(* IEC 61131-3 sources: POMIRTS_lab3/AS/Library/LoopConR/V2.80.0, 3 files *)

(* ---- LoopConR.typ ---- *)
TYPE
	lcrCurveByPoints_TabEntry_type : 	STRUCT
		x : REAL;
		y : REAL;
	END_STRUCT;
	lcrdblpid_par_typ : 	STRUCT
		Y_max : REAL;
		Y_min : REAL;
		K_fact : INT;
		Kp : REAL;
		Tn : REAL;
		Tv : REAL;
	END_STRUCT;
	lcrdblpid_tune_typ : 	STRUCT
		P1_manualAdjust : INT;
		I1_manualAdjust : INT;
		D1_manualAdjust : INT;
		P2_manualAdjust : INT;
		I2_manualAdjust : INT;
		D2_manualAdjust : INT;
		X_min : REAL;
		X_max : REAL;
		X0 : REAL;
		de_min : REAL;
		Y0 : REAL;
		Y1step : REAL;
		Y2step : REAL;
		tuneY1_opt : UDINT;
		tuneY2_opt : UDINT;
		tune_first : USINT;
		hyst : REAL;
		measDelta : REAL;
		osc_opt : lcrpid_tune_osc_options_typ;
		step_opt : lcrpid_tune_step_options_typ;
	END_STRUCT;
	lcrpid_internal_typ : 	STRUCT
		size : UINT;
		valid : BOOL;
		WX_max : REAL;
		WX_min : REAL;
		invert : BOOL;
		deadband : REAL;
		deadband_mode : USINT;
		dY_max : REAL;
		Kp : REAL;
		Kp_Tn : REAL;
		Tv_Tf : REAL;
		Tf_reciproc : REAL;
		Kw : REAL;
		Kfbk_Kp : REAL;
		Kfbk_Kp_max : REAL;
		fbk_mode : USINT;
		d_mode : USINT;
		force_mode : USINT;
		Y_force : REAL;
		W : REAL;
		X : REAL;
		pid_init : USINT;
		Yp1 : DINT;
		Yp2 : DINT;
		dYi1 : DINT;
		dYi2 : DINT;
		Yi1 : DINT;
		Yi2 : DINT;
		dt_Tf : REAL;
		a11 : DINT;
		a12 : DINT;
		a21 : DINT;
		a22 : DINT;
		Yd1 : DINT;
		Yd2 : DINT;
		Ytotal1 : DINT;
		Ytotal2 : DINT;
		Ylim1 : DINT;
		Ylim2 : DINT;
		Y1 : DINT;
		Y2 : DINT;
		deltaY_fbk : REAL;
		e_fbk : REAL;
	END_STRUCT;
	lcrpid_old_typ : 	STRUCT
		processPar : lcrpid_procPar_typ;
		P_manualAdjust : INT;
		I_manualAdjust : INT;
		D_manualAdjust : INT;
		Y_min : REAL;
		Y_max : REAL;
		dY_max : REAL;
		Tf_Tv : REAL;
		Kw : REAL;
		Kfbk : REAL;
		deadband : REAL;
		W : REAL;
		request : UDINT;
		fbk_mode : USINT;
		d_mode : USINT;
		invert : BOOL;
		enable : BOOL;
	END_STRUCT;
	lcrpid_osc_per_typ : 	STRUCT
		max : lcrpid_osc_val_typ;
		min : lcrpid_osc_val_typ;
	END_STRUCT;
	lcrpid_osc_val_typ : 	STRUCT
		X : REAL;
		t : REAL;
	END_STRUCT;
	lcrpid_procPar_typ : 	STRUCT
		size : UINT;
		valid : BOOL;
		stepResp_valid : BOOL;
		stepResp_v : REAL;
		stepResp_t_u : REAL;
		stepResp_t_g : REAL;
		osc_valid : BOOL;
		osc_amplitudeRatio : REAL;
		osc_tPeriod : REAL;
		force_params : BOOL;
		Kp : REAL;
		Kp_tune : REAL;
		Tn : REAL;
		Tn_tune : REAL;
		Tv : REAL;
		Tv_tune : REAL;
	END_STRUCT;
	lcrpid_tune_addpar_typ : 	STRUCT
		t_max_tune : REAL;
		WX_min : REAL;
		WX_max : REAL;
		dY_max : REAL;
		Tf_Tv : REAL;
		Kw : REAL;
		Kfbk : REAL;
		fbk_mode : USINT;
		d_mode : USINT;
		deadband : REAL;
		deadband_mode : USINT;
		invert : BOOL;
	END_STRUCT;
	lcrpid_tune_osc_options_typ : 	STRUCT
		osc_minAmplitude : REAL;
		Q_min : REAL;
	END_STRUCT;
	lcrpid_tune_osc_typ : 	STRUCT
		options : lcrpid_tune_osc_options_typ;
		oscPhase : UINT;
		dir : SINT;
		enHi : BOOL;
		enLo : BOOL;
		Y_hi : REAL;
		Y_lo : REAL;
		i_maxPeriod : UINT;
		i_period : UINT;
		X_ampl : REAL;
		X_avg : REAL;
		X_min_avg : REAL;
		X_max_avg : REAL;
		Y_avg : REAL;
		deltaY : REAL;
		t_Ylohi : ARRAY[0..4] OF REAL;
		t_Yhilo : ARRAY[0..4] OF REAL;
		Q_act : REAL;
		a_wx : REAL;
		amplitudeRatio : REAL;
		Ku : REAL;
		tPeriod : REAL;
		period : ARRAY[0..4] OF lcrpid_osc_per_typ;
	END_STRUCT;
	lcrpid_tune_step_options_typ : 	STRUCT
		eqDeltaX : REAL;
		eqDeltaWX : REAL;
		eqDeltat : REAL;
		evalDeltaX : REAL;
		evalNfilter : UINT;
		exitNotMaxdXCount : UINT;
		exitdXRatio : REAL;
	END_STRUCT;
	lcrpid_tune_step_typ : 	STRUCT
		options : lcrpid_tune_step_options_typ;
		Y0 : REAL;
		Y1 : REAL;
		t_jump : REAL;
		W : REAL;
		X0 : REAL;
		Xmax : REAL;
		Xmin : REAL;
		Xfiltered : REAL;
		deltaXok : BOOL;
		deltaWXok : BOOL;
		eqTime : REAL;
		dir : SINT;
		deltaX : REAL;
		X1 : REAL;
		t1 : REAL;
		t1set : BOOL;
		dX_dt : REAL;
		dX_dt_max : REAL;
		XmaxGrad : REAL;
		maxX1 : REAL;
		maxX2 : REAL;
		maxt1 : REAL;
		maxt2 : REAL;
		tmaxGrad : REAL;
		gainFactor : REAL;
		deadTime : REAL;
		riseTime : REAL;
		notMaxCount : UINT;
		gradientRatio : REAL;
	END_STRUCT;
	lcrpt2o_Internal_typ : 	STRUCT
		Ts : DINT;
		Ts_dbl_1 : UDINT;
		Ts_dbl_2 : UDINT;
		V_old : REAL;
		D_old : REAL;
		Tf_old : REAL;
		Set_y_old : USINT;
		Set_y_2 : USINT;
		x1_dbl_1 : UDINT;
		x1_dbl_2 : UDINT;
		x2_dbl_1 : UDINT;
		x2_dbl_2 : UDINT;
		Sqrt_D_1_dbl_1 : UDINT;
		Sqrt_D_1_dbl_2 : UDINT;
		Ts_Tf_dbl_1 : UDINT;
		Ts_Tf_dbl_2 : UDINT;
		Exp_D_Ts_Tf_dbl_1 : UDINT;
		Exp_D_Ts_Tf_dbl_2 : UDINT;
		a0_dbl_1 : UDINT;
		a0_dbl_2 : UDINT;
		a1_dbl_1 : UDINT;
		a1_dbl_2 : UDINT;
		b0_dbl_1 : UDINT;
		b0_dbl_2 : UDINT;
		b1_dbl_1 : UDINT;
		b1_dbl_2 : UDINT;
		Bootkey : UDINT;
	END_STRUCT;
	lcrschedule_add_typ : 	STRUCT
		periodTime : REAL;
		onTime : REAL;
		t_on_intern : REAL;
		bcOnTime : REAL;
		sortIndex : UINT;
		fbkPWM : LCRPWM;
		flagDelay : BOOL;
	END_STRUCT;
	lcrschedule_par_typ : 	STRUCT
		P : REAL;
		X : REAL;
		pulse : BOOL;
		Pout : REAL;
		lim : BOOL;
		Internal : lcrschedule_add_typ;
	END_STRUCT;
	lcrslimpid_par_typ : 	STRUCT
		Y_max : REAL;
		Y_min : REAL;
		Kp : REAL;
		Tn : REAL;
		Tv : REAL;
		Kfbk : REAL;
	END_STRUCT;
	lcrtemp_add_typ : 	STRUCT
		mem01 : REAL;
		mem02 : REAL;
		mem10 : REAL;
		mem20 : REAL;
		exp_mem : REAL;
		cnt01 : REAL;
		cnt02 : REAL;
		cnt10 : REAL;
		cnt20 : REAL;
		cnt03 : REAL;
		cnt30 : REAL;
		cnt00 : REAL;
		t_ignore_dT_heat : REAL;
		t_ignore_dT_free : REAL;
		t_ignore_dT_cool : REAL;
		yMin : REAL;
		yMax : REAL;
		reserved3 : UDINT;
		reserved4 : UDINT;
		reserved5 : BOOL;
		reserved6 : BOOL;
	END_STRUCT;
	lcrtemp_pid_internal_typ : 	STRUCT
		enable_cooling : BOOL;
		disable_heating : BOOL;
		hyst : REAL;
		delay : REAL;
		Kw : REAL;
		Kfbk : REAL;
		Kp_h : REAL;
		Tn_h : REAL;
		Tv_h : REAL;
		Kp_c : REAL;
		Tn_c : REAL;
		Tv_c : REAL;
		dynGeneral : REAL;
		dynHeat : REAL;
		dynCool : REAL;
		mem01 : REAL;
		mem02 : REAL;
		mem10 : REAL;
		mem20 : REAL;
		exp_mem : REAL;
		yMin : REAL;
		yMax : REAL;
	END_STRUCT;
	lcrtemp_pid_opt_typ : 	STRUCT
		Kp_h : REAL;
		Tn_h : REAL;
		Tv_h : REAL;
		Kp_c : REAL;
		Tn_c : REAL;
		Tv_c : REAL;
		dynGeneral : REAL;
		dynHeat : REAL;
		dynCool : REAL;
	END_STRUCT;
	lcrtemp_pid_set_typ : 	STRUCT
		hyst : REAL;
		delay : REAL;
		Kw : REAL;
		Kfbk : REAL;
	END_STRUCT;
	lcrtemp_set_typ : 	STRUCT
		enable_cooling : BOOL;
		disable_heating : BOOL;
		PIDpara : lcrtemp_pid_opt_typ;
		TuneSet : lcrtemp_tune_set_typ;
		PIDSet : lcrtemp_pid_set_typ;
		Internal : lcrtemp_add_typ;
	END_STRUCT;
	lcrtemp_tune_internal_typ : 	STRUCT
		cool_tuning : BOOL;
		disable_heating : BOOL;
		mode : UDINT;
		Temp_amb : REAL;
		dRatio_heat : REAL;
		cnt_tp_heat : REAL;
		delta_T_heat : REAL;
		dT_min_heat : REAL;
		dRatio_free : REAL;
		cnt_tp_free : REAL;
		delta_T_free : REAL;
		dT_min_free : REAL;
		dRatio_cool : REAL;
		cnt_tp_cool : REAL;
		delta_T_cool : REAL;
		dT_min_cool : REAL;
		delta_T_sync_heat : REAL;
		delta_dT_sync_heat : REAL;
		cnt_wait_heat : REAL;
		delta_T_sync_free : REAL;
		delta_dT_sync_free : REAL;
		cnt_wait_free : REAL;
		delta_T_sync_cool : REAL;
		delta_dT_sync_cool : REAL;
		cnt_wait_cool : REAL;
		filter_base_T : REAL;
		t_ignore_dT_heat : REAL;
		t_ignore_dT_free : REAL;
		t_ignore_dT_cool : REAL;
		delta_T_sync_stop : REAL;
	END_STRUCT;
	lcrtemp_tune_set_typ : 	STRUCT
		mode : UDINT;
		Temp_amb : REAL;
		dRatio_heat : REAL;
		cnt_tp_heat : REAL;
		delta_T_heat : REAL;
		dT_min_heat : REAL;
		dRatio_free : REAL;
		cnt_tp_free : REAL;
		delta_T_free : REAL;
		dT_min_free : REAL;
		dRatio_cool : REAL;
		cnt_tp_cool : REAL;
		delta_T_cool : REAL;
		dT_min_cool : REAL;
		delta_T_sync_heat : REAL;
		delta_dT_sync_heat : REAL;
		cnt_wait_heat : REAL;
		delta_T_sync_free : REAL;
		delta_dT_sync_free : REAL;
		cnt_wait_free : REAL;
		delta_T_sync_cool : REAL;
		delta_dT_sync_cool : REAL;
		cnt_wait_cool : REAL;
		filter_base_T : REAL;
		delta_T_sync_stop : REAL;
		Y_heat_tune : REAL;
	END_STRUCT;
END_TYPE

(* ---- LoopConR.fun ---- *)
FUNCTION_BLOCK LCRPID
	VAR_INPUT
		enable : BOOL;
		ident : UDINT;
		W : REAL;
		X : REAL;
		Y_max : REAL;
		Y_min : REAL;
		A : REAL;
		Y_man : REAL;
		Y_fbk : REAL;
		hold_I : BOOL;
		mode : USINT;
	END_VAR
	VAR_OUTPUT
		status : UINT;
		e : REAL;
		Y : REAL;
		Yp : REAL;
		Yi : REAL;
		Yd : REAL;
	END_VAR
	VAR
		Set_Yi : BOOL;
		Yi_set : REAL;
		force_Yi : BOOL;
		Yi_min : REAL;
		Yi_max : REAL;
		joltFreeDoneLowerLim : BOOL;
		joltFreeDoneUpperLim : BOOL;
		Yi_minInternal : REAL;
		Yi_maxInternal : REAL;
		Tv_Tf_old : REAL;
		enable_old : BOOL;
		e_old : REAL;
		deadband_state : UINT;
		sysinfo_inst : SysInfo;
		scal_inst : LCRScal;
		store1 : UDINT;
		store2 : UDINT;
		timeCnt : UDINT;
		musecs_old : UINT;
	END_VAR
END_FUNCTION_BLOCK

FUNCTION_BLOCK LCRScal
	VAR_INPUT
		x : REAL;
		x1 : REAL;
		y1 : REAL;
		x2 : REAL;
		y2 : REAL;
	END_VAR
	VAR_OUTPUT
		y : REAL;
	END_VAR
END_FUNCTION_BLOCK

FUNCTION_BLOCK LCRCurveByPoints
	VAR_INPUT
		x : REAL;
		NoOfPoints : UINT;
		ptr_table : REFERENCE TO lcrCurveByPoints_TabEntry_type;
	END_VAR
	VAR_OUTPUT
		status : UINT;
		y : REAL;
	END_VAR
	VAR
		i_tab : INT;
		iterations : UINT;
		scal1 : LCRScal;
	END_VAR
END_FUNCTION_BLOCK

FUNCTION_BLOCK LCRPIDpara
	VAR_INPUT
		enable : BOOL;
		enter : BOOL;
		WX_max : REAL;
		WX_min : REAL;
		invert : BOOL;
		deadband : REAL;
		deadband_mode : USINT;
		dY_max : REAL;
		Kp : REAL;
		Tn : REAL;
		Tv : REAL;
		Tf : REAL;
		Kw : REAL;
		Kfbk : REAL;
		fbk_mode : USINT;
		d_mode : USINT;
	END_VAR
	VAR_OUTPUT
		status : UINT;
		ident : UDINT;
	END_VAR
	VAR
		internal_data : lcrpid_internal_typ;
	END_VAR
END_FUNCTION_BLOCK

FUNCTION_BLOCK LCRContinServo
	VAR_INPUT
		enable : BOOL;
		x : REAL;
		max_value : REAL;
		min_value : REAL;
		t_impulse : REAL;
		t_change_up : REAL;
		t_change_down : REAL;
		ref : BOOL;
	END_VAR
	VAR_OUTPUT
		status : UINT;
		up : BOOL;
		down : BOOL;
		hysteresis_up : REAL;
		hysteresis_down : REAL;
		refOk : BOOL;
	END_VAR
	VAR
		enable_old : BOOL;
		counter_state : UINT;
		bootkey_old : UDINT;
		systicks_old : UDINT;
		musecs_old : UINT;
		ref_old : BOOL;
		t_cnt_1 : DINT;
		t_cnt_2 : DINT;
		y_dbl_1 : DINT;
		y_dbl_2 : DINT;
		sysInfo_inst : SysInfo;
	END_VAR
END_FUNCTION_BLOCK

FUNCTION_BLOCK LCRPT1
	VAR_INPUT
		enable : BOOL;
		x : REAL;
		t : REAL;
		y_set : REAL;
		set : BOOL;
	END_VAR
	VAR_OUTPUT
		status : UINT;
		y : REAL;
	END_VAR
	VAR
		counter_state : UINT;
		bootkey_old : UDINT;
		systicks_old : UDINT;
		musecs_old : UINT;
		y_dbl_1 : DINT;
		y_dbl_2 : DINT;
		sysinfo_inst : SysInfo;
	END_VAR
END_FUNCTION_BLOCK

FUNCTION_BLOCK LCRRamp
	VAR_INPUT
		enable : BOOL;
		x : REAL;
		dy_up : REAL;
		dy_down : REAL;
		y_max : REAL;
		y_min : REAL;
		y_set : REAL;
		set : BOOL;
	END_VAR
	VAR_OUTPUT
		status : UINT;
		y : REAL;
		x_reached : BOOL;
		max_limit : BOOL;
		min_limit : BOOL;
	END_VAR
	VAR
		y_dbl_1 : DINT;
		y_dbl_2 : DINT;
		timestore1 : UDINT;
		timestore2 : UDINT;
		getDtForceOff : UDINT;
		sysinfo_inst : SysInfo;
	END_VAR
END_FUNCTION_BLOCK

FUNCTION_BLOCK LCRIntegrate
	VAR_INPUT
		enable : BOOL;
		x : REAL;
		tn : REAL;
		y_max : REAL;
		y_min : REAL;
		y_set : REAL;
		set : BOOL;
	END_VAR
	VAR_OUTPUT
		status : UINT;
		y : REAL;
		max_limit : BOOL;
		min_limit : BOOL;
	END_VAR
	VAR
		counter_state : UINT;
		bootkey_old : UDINT;
		systicks_old : UDINT;
		musecs_old : UINT;
		y_dbl_1 : DINT;
		y_dbl_2 : DINT;
		sysinfo_inst : SysInfo;
	END_VAR
END_FUNCTION_BLOCK

FUNCTION_BLOCK LCRLimit
	VAR_INPUT
		in : REAL;
		max_value : DINT;
		min_value : DINT;
	END_VAR
	VAR_OUTPUT
		status : UINT;
		out : DINT;
		max_limit : BOOL;
		min_limit : BOOL;
	END_VAR
END_FUNCTION_BLOCK

FUNCTION_BLOCK LCRLimScal
	VAR_INPUT
		x : REAL;
		x1 : REAL;
		y1 : REAL;
		x2 : REAL;
		y2 : REAL;
	END_VAR
	VAR_OUTPUT
		y : REAL;
	END_VAR
END_FUNCTION_BLOCK

FUNCTION_BLOCK LCRPWM
	VAR_INPUT
		enable : BOOL;
		x : REAL;
		max_value : REAL;
		min_value : REAL;
		t_min_pulse : REAL;
		t_period : REAL;
	END_VAR
	VAR_OUTPUT
		status : UINT;
		pulse : BOOL;
		t_on : REAL;
		t_off : REAL;
	END_VAR
	VAR
		cnt_terron_1 : DINT;
		cnt_terron_2 : DINT;
		cnt_terroff_1 : DINT;
		cnt_terroff_2 : DINT;
		cnt_t_pulse_1 : DINT;
		cnt_t_pulse_2 : DINT;
		store1 : UDINT;
		store2 : UDINT;
		timeCnt : UDINT;
		sysinfo_inst : SysInfo;
		corr : BOOL;
	END_VAR
END_FUNCTION_BLOCK

FUNCTION_BLOCK LCRMovAvgFlt
	VAR_INPUT
		enable : BOOL;
		x : REAL;
		base : UINT;
	END_VAR
	VAR_OUTPUT
		status : UINT;
		y : REAL;
	END_VAR
	VAR
		sum_old_dbl_1 : DINT;
		sum_old_dbl_2 : DINT;
		x_old : ARRAY[0..31] OF REAL;
		p_xold : UDINT;
		i_xold : UINT;
		base_old : UINT;
		enable_old : BOOL;
		bootkey_old : UDINT;
	END_VAR
END_FUNCTION_BLOCK

FUNCTION_BLOCK LCRTimeBasedOnOff
	VAR_INPUT
		enable : BOOL;
		x : REAL;
		max_value : REAL;
		min_value : REAL;
		timpulse : REAL;
		tchange_up : REAL;
		tchange_down : REAL;
		ref : BOOL;
	END_VAR
	VAR_OUTPUT
		status : UINT;
		up : BOOL;
		down : BOOL;
		hysteresis_up : REAL;
		hysteresis_down : REAL;
		refOk : BOOL;
	END_VAR
	VAR
		enable_old : BOOL;
		counter_state : UINT;
		bootkey_old : UDINT;
		systicks_old : UDINT;
		musecs_old : UINT;
		ref_old : BOOL;
		t_cnt_1 : DINT;
		t_cnt_2 : DINT;
		y_dbl_1 : DINT;
		y_dbl_2 : DINT;
		sysInfo_inst : SysInfo;
	END_VAR
END_FUNCTION_BLOCK

FUNCTION_BLOCK LCRDifferentiate
	VAR_INPUT
		enable : BOOL;
		x : REAL;
		tv : REAL;
		tf : REAL;
	END_VAR
	VAR_OUTPUT
		status : UINT;
		y : REAL;
	END_VAR
	VAR
		store1 : UDINT;
		store2 : UDINT;
		timeCnt : UDINT;
		counter_state : UINT;
		bootkey_old : UDINT;
		systicks_old : UDINT;
		musecs_old : UINT;
		sysinfo_inst : SysInfo;
		a11 : DINT;
		a12 : DINT;
		a21 : DINT;
		a22 : DINT;
	END_VAR
END_FUNCTION_BLOCK

FUNCTION_BLOCK LCRSlimPID
	VAR_INPUT
		enable : BOOL;
		W : REAL;
		X : REAL;
		request : UDINT;
		pPar : REFERENCE TO lcrslimpid_par_typ;
	END_VAR
	VAR_OUTPUT
		e : REAL;
		Y : REAL;
		status : UINT;
		addInfo : UINT;
	END_VAR
	VAR
		MovAvgFlt_inst : LCRMovAvgFlt;
		PIDTune_inst : LCRPIDTune;
		PID_inst : LCRPID;
		enable_old : BOOL;
		requ_old : UDINT;
	END_VAR
END_FUNCTION_BLOCK

FUNCTION_BLOCK LCRPIDTune
	VAR_INPUT
		enable : BOOL;
		Y_min : REAL;
		Y_max : REAL;
		Y0 : REAL;
		Y1 : REAL;
		okToStep : BOOL;
		X0 : REAL;
		X_min : REAL;
		X_max : REAL;
		P_manualAdjust : INT;
		I_manualAdjust : INT;
		D_manualAdjust : INT;
		request : UDINT;
		pAddPar : REFERENCE TO lcrpid_tune_addpar_typ;
		pOptions_osc : REFERENCE TO lcrpid_tune_osc_options_typ;
		pOptions_step : REFERENCE TO lcrpid_tune_step_options_typ;
	END_VAR
	VAR_OUTPUT
		status : UINT;
		addInfo : UINT;
		ident : UDINT;
		state : UINT;
		rdyToStep : BOOL;
	END_VAR
	VAR
		t_autotune : REAL;
		status_tmp : UINT;
		counter_state : UINT;
		bootkey_old : UDINT;
		systicks_old : UDINT;
		musecs_old : UINT;
		curveDown : BOOL;
		e : REAL;
		e_minAmp : REAL;
		e_old_up : REAL;
		e_old_down : REAL;
		curveUp : BOOL;
		e_old : REAL;
		sysinfo_inst : SysInfo;
		MovAvgFlt_inst : LCRMovAvgFlt;
		old : lcrpid_old_typ;
		processPar : lcrpid_procPar_typ;
		internal_data : lcrpid_internal_typ;
		addPar : lcrpid_tune_addpar_typ;
		oscillation : lcrpid_tune_osc_typ;
		stepresponse : lcrpid_tune_step_typ;
	END_VAR
END_FUNCTION_BLOCK

FUNCTION_BLOCK LCRPFM
	VAR_INPUT
		enable : BOOL;
		x : REAL;
		max_value : REAL;
		min_value : REAL;
		t_pulse : REAL;
		t_pause : REAL;
	END_VAR
	VAR_OUTPUT
		status : UINT;
		pulse : BOOL;
	END_VAR
	VAR
		area : REAL;
		area_c : REAL;
		range : REAL;
		last : REAL;
		tpls : REAL;
		enable_old : BOOL;
		counter_state : UINT;
		bootkey_old : UDINT;
		systicks_old : UDINT;
		musecs_old : UINT;
		sysinfo_inst : SysInfo;
	END_VAR
END_FUNCTION_BLOCK

FUNCTION_BLOCK LCRSimModExt
	VAR_INPUT
		enable : BOOL;
		Tt_h : DINT;
		Tt_c : DINT;
		k_h : REAL;
		k_c : REAL;
		PT2_T1 : REAL;
		PT2_T2 : REAL;
		Temp_amb : REAL;
		Temp_c : REAL;
		Alpha_h : REAL;
		Alpha_c : REAL;
	END_VAR
	VAR_OUTPUT
		y : REAL;
		status : UINT;
	END_VAR
	VAR
		Tt_heat : LCRTt;
		Tt_cool : LCRTt;
		k_h_intern : REAL;
		k_c_intern : REAL;
		PT2 : LCRPT2;
		y_c : REAL;
		y_end : REAL;
		y_h : REAL;
		Bootkey : UDINT;
		enable_old : BOOL;
	END_VAR
END_FUNCTION_BLOCK

FUNCTION_BLOCK LCRTt
	VAR_INPUT
		enable : BOOL;
		Tt : DINT;
		x : REAL;
		y_set : REAL;
		set : BOOL;
	END_VAR
	VAR_OUTPUT
		y : REAL;
		status : UINT;
	END_VAR
	VAR
		Ts : DINT;
		Tt_Max : DINT;
		pRingBuf : REFERENCE TO REAL;
		pBuf_OutIn : REFERENCE TO REAL;
		set_old : USINT;
		Set_y : USINT;
		enable_old : BOOL;
		Bootkey : UDINT;
	END_VAR
END_FUNCTION_BLOCK

FUNCTION_BLOCK LCRPT2
	VAR_INPUT
		enable : BOOL;
		V : REAL;
		T1 : REAL;
		T2 : REAL;
		x : REAL;
		y_set : REAL;
		set : USINT;
	END_VAR
	VAR_OUTPUT
		y : REAL;
		status : UINT;
	END_VAR
	VAR
		x1_dbl_1 : UDINT;
		x1_dbl_2 : UDINT;
		x2_dbl_1 : UDINT;
		x2_dbl_2 : UDINT;
		Ts : DINT;
		Ts_dbl_1 : UDINT;
		Ts_dbl_2 : UDINT;
		set_old : USINT;
		Set_y : USINT;
		Bootkey : UDINT;
	END_VAR
END_FUNCTION_BLOCK

FUNCTION_BLOCK LCRPT1e
	VAR_INPUT
		enable : BOOL;
		V : REAL;
		T1 : REAL;
		x : REAL;
		y_set : REAL;
		set : USINT;
	END_VAR
	VAR_OUTPUT
		y : REAL;
		status : UINT;
	END_VAR
	VAR
		x1_dbl_1 : UDINT;
		x1_dbl_2 : UDINT;
		Ts : DINT;
		Ts_dbl_1 : UDINT;
		Ts_dbl_2 : UDINT;
		set_old : USINT;
		Set_y : USINT;
		Bootkey : UDINT;
	END_VAR
END_FUNCTION_BLOCK

FUNCTION_BLOCK LCRDblActPID
	VAR_INPUT
		enable : BOOL;
		W : REAL;
		X : REAL;
		Y_man : REAL;
		hold_I : BOOL;
		mode : USINT;
		okToStep : BOOL;
		pPar1 : REFERENCE TO lcrdblpid_par_typ;
		pPar2 : REFERENCE TO lcrdblpid_par_typ;
		pAddPar : REFERENCE TO lcrpid_tune_addpar_typ;
		pOpt : REFERENCE TO lcrdblpid_tune_typ;
	END_VAR
	VAR_OUTPUT
		e : REAL;
		Y1 : REAL;
		Y2 : REAL;
		status : UINT;
		tuneState : USINT;
		rdyToStep : BOOL;
	END_VAR
	VAR
		enable_old : BOOL;
		pid : LCRPID;
		tune : LCRPIDTune;
		sysinfo_inst : SysInfo;
		gradient : REAL;
		Y_avg : REAL;
		tcnt_1 : UDINT;
		tcnt_2 : UDINT;
		Tmeas : REAL;
		y_lim_old : REAL;
		p_fact : REAL;
		bootkey_old : UDINT;
		systicks_old : UDINT;
		musecs_old : UINT;
		use_par : USINT;
		meas : USINT;
		mode_old : USINT;
		tune_step : USINT;
		tune_grad : USINT;
		tune_2nd : USINT;
		invert : USINT;
		counter_state : USINT;
		mode_int : USINT;
	END_VAR
END_FUNCTION_BLOCK

FUNCTION_BLOCK LCRMinMax
	VAR_INPUT
		reset : BOOL;
		in : REAL;
	END_VAR
	VAR_OUTPUT
		out_min : REAL;
		out_max : REAL;
	END_VAR
END_FUNCTION_BLOCK

FUNCTION_BLOCK LCRTempPID
	VAR_INPUT
		enable : BOOL;
		Temp_set : REAL;
		Temp : REAL;
		Y_man : REAL;
		mode : UDINT;
		update : BOOL;
		pSettings : REFERENCE TO lcrtemp_set_typ;
	END_VAR
	VAR_OUTPUT
		y_heat : REAL;
		y_cool : REAL;
		status : UINT;
	END_VAR
	VAR
		pid : LCRPID;
		pid_para : LCRPIDpara;
		Temp_set_delay : REAL;
		Temp_set_int : REAL;
		TempSetOld : REAL;
		delayCnt : REAL;
		delayFlag : BOOL;
		enable_old : BOOL;
		stateOld : SINT;
		state : SINT;
		a : REAL;
		sysinfo_inst : SysInfo;
		para_check_done : USINT;
		internal_para : lcrtemp_pid_internal_typ;
		dbl_dt : REAL;
		tAlt : REAL;
		altTime : REAL;
		tKnick : REAL;
		fAlt : REAL;
		altActive : BOOL;
		a_alt : REAL;
		a_e : REAL;
		a_internal : REAL;
		err_flag : BOOL;
		Temp_set_int_old1 : REAL;
		Temp_set_int_old2 : REAL;
		Temp_set_int_old3 : REAL;
		mode_old : UDINT;
		timestore1 : UDINT;
		timestore2 : UDINT;
		yManInternal : REAL;
		timeCnt : UDINT;
	END_VAR
END_FUNCTION_BLOCK

FUNCTION_BLOCK LCRTempTune
	VAR_INPUT
		enable : BOOL;
		start : BOOL;
		Temp_set : REAL;
		Temp : REAL;
		okToHeat : BOOL;
		okToFree : BOOL;
		okToFreeEnd : BOOL;
		okToCool : BOOL;
		okToCoolEnd : BOOL;
		pSettings : REFERENCE TO lcrtemp_set_typ;
	END_VAR
	VAR_OUTPUT
		y_heat : REAL;
		y_cool : REAL;
		rdyToHeat : BOOL;
		rdyToFree : BOOL;
		rdyToFreeEnd : BOOL;
		rdyToCool : BOOL;
		rdyToCoolEnd : BOOL;
		done : BOOL;
		busy : BOOL;
		status : UINT;
	END_VAR
	VAR
		enable_old : BOOL;
		pid : LCRPID;
		pid_para : LCRPIDpara;
		DT2 : LCRDifferentiate;
		pt2 : LCRPT2o;
		Temp_flt : REAL;
		step : UINT;
		t : REAL;
		Temp_start : REAL;
		mem00 : REAL;
		cnt02 : REAL;
		cnt33 : REAL;
		cnt20 : REAL;
		pem01 : REAL;
		pem33 : REAL;
		pem10 : REAL;
		pem02 : REAL;
		pem44 : REAL;
		pem20 : REAL;
		tol01 : REAL;
		tol10 : REAL;
		tol02 : REAL;
		tol20 : REAL;
		tol22 : REAL;
		Temp_old : REAL;
		delta_Temp : REAL;
		tcnt_1 : UDINT;
		tcnt_2 : UDINT;
		tcnt_dT_1 : UDINT;
		tcnt_dT_2 : UDINT;
		sysinfo_inst : SysInfo;
		Temp_set_internal : REAL;
		timecounter : REAL;
		internal_para : lcrtemp_tune_internal_typ;
		dbl_dt : REAL;
		call_counter : UDINT;
		store1 : UDINT;
		store2 : UDINT;
		timeCnt : UDINT;
		timer2 : REAL;
		waitCounter : UINT;
		Y_heat_tune_intern : REAL;
	END_VAR
END_FUNCTION_BLOCK

FUNCTION_BLOCK LCRPT2o (* Oscillating 2nd order delay element. *)
	VAR_INPUT
		enable : BOOL;
		V : REAL;
		D : REAL;
		Tf : REAL;
		u : REAL;
		Set_y : USINT;
		y_set : REAL;
	END_VAR
	VAR_OUTPUT
		y : REAL;
		status : UINT;
	END_VAR
	VAR
		Internal : lcrpt2o_Internal_typ;
	END_VAR
END_FUNCTION_BLOCK

FUNCTION_BLOCK LCRSchedulePWM
	VAR_INPUT
		enable : BOOL;
		Pmax : REAL;
		n : UINT;
		pPar : UDINT;
		min_value : REAL;
		max_value : REAL;
		t_min_pulse : REAL;
		t_period : REAL;
	END_VAR
	VAR_OUTPUT
		status : UINT;
	END_VAR
	VAR
		sysinfo_inst : SysInfo;
		store1 : UDINT;
		store2 : UDINT;
		timeCnt : UDINT;
		numberUnits : UINT;
		limFact : UINT;
		enable_old : BOOL;
		cmd_delay : BOOL;
		err_flag : BOOL;
		limAll : BOOL;
		Pact : REAL;
		Pman : REAL;
		intern0 : ARRAY[0..5] OF REAL;
		in : REFERENCE TO lcrschedule_par_typ;
	END_VAR
END_FUNCTION_BLOCK

(* ---- LoopConR.var ---- *)
VAR CONSTANT
	LCR_ERR_DISABLED : UINT := 65534;
	LCR_ERR_LCRContinServo_TCHANGE : UINT := 12035;
	LCR_ERR_LCRContinServo_TIMPULSE : UINT := 12036;
	LCR_ERR_LCRCurveByPoints_TABLE : UINT := 12045;
	LCR_ERR_LCRDBLPID_DX_DT : UINT := 31562;
	LCR_ERR_LCRDBLPID_WX_LOW : UINT := 31561;
	LCR_ERR_LCRIntegrate_TN : UINT := 31550;
	LCR_ERR_LCRMovAvgFlt_BASE : UINT := 31551;
	LCR_ERR_LCRPID_IDENT : UINT := 31552;
	LCR_ERR_LCRPID_MODE : UINT := 31553;
	LCR_ERR_LCRPID_PAR_DEADBAND : UINT := 12044;
	LCR_ERR_LCRPID_PAR_DEADBAND_MODE : UINT := 12042;
	LCR_ERR_LCRPID_PAR_DMODE : UINT := 31556;
	LCR_ERR_LCRPID_PAR_DYMAX : UINT := 31557;
	LCR_ERR_LCRPID_PAR_FBKMODE : UINT := 31558;
	LCR_ERR_LCRPID_PAR_KFBK : UINT := 12025;
	LCR_ERR_LCRPID_PAR_KP : UINT := 12026;
	LCR_ERR_LCRPID_PAR_KW : UINT := 12027;
	LCR_ERR_LCRPID_PAR_TF : UINT := 12028;
	LCR_ERR_LCRPID_PAR_TN : UINT := 12029;
	LCR_ERR_LCRPID_PAR_TV : UINT := 12030;
	LCR_ERR_LCRPID_PAR_WX_MAXMIN : UINT := 12043;
	LCR_ERR_LCRPID_PARADAT : UINT := 31554;
	LCR_ERR_LCRPIDTune_ABORT : UINT := 12038;
	LCR_ERR_LCRPIDTune_CONTROL_VAR : UINT := 31560;
	LCR_ERR_LCRPIDTune_INVALID_REQU : UINT := 31559;
	LCR_ERR_LCRPIDTune_MAXMIN : UINT := 31564;
	LCR_ERR_LCRPIDTune_PARAMETER : UINT := 12039;
	LCR_ERR_LCRPIDTune_TIMEOUT : UINT := 12040;
	LCR_ERR_LCRPIDTune_W_CHANGED : UINT := 12041;
	LCR_ERR_LCRPT1_T : UINT := 12031;
	LCR_ERR_LCRPT12_T1_NEG : UINT := 12046;
	LCR_ERR_LCRPT12_T2_NEG : UINT := 12047;
	LCR_ERR_LCRPWM_TMINPULSE : UINT := 12032;
	LCR_ERR_LCRPWM_TPERIOD : UINT := 12033;
	LCR_ERR_LCRRamp_DYUP_DYDOWN : UINT := 12034;
	LCR_ERR_LCRTEMPPID_ILLEGALMODE : UINT := 31569;
	LCR_ERR_LCRTEMPPID_INVALID_MODE : UINT := 33151;
	LCR_ERR_LCRTEMPPID_NO_TALT : UINT := 31572;
	LCR_ERR_LCRTEMPPID_TKNICK : UINT := 31571;
	LCR_ERR_LCRTEMPPID_WR_PARA : UINT := 31567;
	LCR_ERR_LCRTEMPPID_WR_PTR : UINT := 31568;
	LCR_ERR_LCRTEMPTune_DT_IGNORED : UINT := 33152;
	LCR_ERR_LCRTEMPTune_INVALID_MODE : UINT := 33150;
	LCR_ERR_LCRTEMPTune_TASKTIME_0 : UINT := 31570;
	LCR_ERR_LCRTEMPTune_WR_PTR : UINT := 31566;
	LCR_ERR_LCRTEMPTune_WR_TSET : UINT := 31567;
	LCR_ERR_LCRTT_TT_NEG : UINT := 12048;
	LCR_ERR_MAXMIN : UINT := 12037;
	LCR_ERR_POINTER : UINT := 31563;
	LCR_ERR_PT2O_D_NEG : UINT := 33153;
	LCR_ERR_PT2O_TF_NEG_ZERO : UINT := 33154;
	LCR_ERR_SCHEDULE_N : UINT := 31574;
	LCR_ERR_SCHEDULE_P : UINT := 31573;
	LCR_ERROR : UINT := 12025;
	LCR_WARN_LCRDBLPID_TUNE_CHANGE : UINT := 12019;
	LCR_WARN_LCRPID_A_LIMIT : UINT := 12008;
	LCR_WARN_LCRPID_I_MAXLIMIT : UINT := 12001;
	LCR_WARN_LCRPID_I_MINLIMIT : UINT := 12002;
	LCR_WARN_LCRPID_YFBK_LIMIT : UINT := 12003;
	LCR_WARN_LCRPID_YMAN_LIMIT : UINT := 12009;
	LCR_WARN_LCRPIDTune_CYCLETIME : UINT := 12004;
	LCR_WARN_LCRPT12_T1_INT : UINT := 12011;
	LCR_WARN_LCRPT12_T1_TS : UINT := 12010;
	LCR_WARN_LCRPT12_T1_ZERO : UINT := 12005;
	LCR_WARN_LCRPT12_T2_INT : UINT := 12014;
	LCR_WARN_LCRPT12_T2_TS : UINT := 12013;
	LCR_WARN_LCRPT12_T2_ZERO : UINT := 12012;
	LCR_WARN_LCRTEMPPID_WR_PARA : UINT := 12024;
	LCR_WARN_LCRTEMPTune_ASYNC : UINT := 33101;
	LCR_WARN_LCRTEMPTune_DT_HIGH : UINT := 33100;
	LCR_WARN_LCRTEMPTune_HEAT_TP : UINT := 12021;
	LCR_WARN_LCRTEMPTune_WR_BASE : UINT := 12023;
	LCR_WARN_LCRTEMPTune_WR_PARA : UINT := 12022;
	LCR_WARN_LCRTT_MEM : UINT := 12018;
	LCR_WARN_LCRTT_TT_INT : UINT := 12017;
	LCR_WARN_LCRTT_TT_TS : UINT := 12016;
	LCR_WARN_LCRTT_TT_ZERO : UINT := 12015;
	LCR_WARN_PT2O_TF_TS : UINT := 33102;
	LCR_WARN_Tx_DT : UINT := 12007;
	LCRDBLPID_MODE_TUNE_4 : USINT := 6;
	LCRDBLPID_MODE_TUNE_6 : USINT := 7;
	LCRDBLPID_MODE_TUNE_Y1 : USINT := 8;
	LCRDBLPID_MODE_TUNE_Y2 : USINT := 9;
	LCRDBLPID_TSTATE_ERROR : USINT := 4;
	LCRDBLPID_TSTATE_FINISHED : USINT := 3;
	LCRDBLPID_TSTATE_OFF : USINT := 0;
	LCRDBLPID_TSTATE_Y1 : USINT := 1;
	LCRDBLPID_TSTATE_Y2 : USINT := 2;
	LCRPID_D_MODE_E : USINT := 2;
	LCRPID_D_MODE_X : USINT := 1;
	LCRPID_DEADBAND_MODE_STANDARD : USINT := 1;
	LCRPID_DEADBAND_MODE_STANDARD_I : USINT := 2;
	LCRPID_DEADBAND_MODE_ZERO : USINT := 0;
	LCRPID_FBK_MODE_EXT_SELECTOR : USINT := 3;
	LCRPID_FBK_MODE_EXTERN : USINT := 2;
	LCRPID_FBK_MODE_INTERN : USINT := 1;
	LCRPID_FBK_MODE_SET_YI : USINT := 5;
	LCRPID_FBK_MODE_LIMIT_YI : USINT := 4;
	LCRPID_MODE_AUTO : USINT := 1;
	LCRPID_MODE_CLOSE : USINT := 4;
	LCRPID_MODE_CLOSE_JOLTFREE : USINT := 104;
	LCRPID_MODE_FREEZE : USINT := 5;
	LCRPID_MODE_FREEZE_JOLTFREE : USINT := 105;
	LCRPID_MODE_MAN : USINT := 2;
	LCRPID_MODE_MAN_JOLTFREE : USINT := 102;
	LCRPID_MODE_OFF : USINT := 0;
	LCRPID_MODE_OPEN : USINT := 3;
	LCRPID_MODE_OPEN_JOLTFREE : USINT := 103;
	LCRPID_TUNE_ADDINFO_OSC_PERIOD : UINT := 111;
	LCRPID_TUNE_REQU_CHR_DIST_AP : UDINT := 1000;
	LCRPID_TUNE_REQU_CHR_DIST_OS : UDINT := 2000;
	LCRPID_TUNE_REQU_CHR_REF_AP : UDINT := 4000;
	LCRPID_TUNE_REQU_CHR_REF_OS : UDINT := 5000;
	LCRPID_TUNE_REQU_DIR_NEG : UDINT := 20;
	LCRPID_TUNE_REQU_DIR_POS : UDINT := 10;
	LCRPID_TUNE_REQU_OFF : UDINT := 0;
	LCRPID_TUNE_REQU_OSC_1 : UDINT := 10000;
	LCRPID_TUNE_REQU_OSC_2 : UDINT := 20000;
	LCRPID_TUNE_REQU_OSC_3 : UDINT := 30000;
	LCRPID_TUNE_REQU_OSCILLATE : UDINT := 1;
	LCRPID_TUNE_REQU_P : UDINT := 300;
	LCRPID_TUNE_REQU_PER_3 : UDINT := 300000;
	LCRPID_TUNE_REQU_PER_4 : UDINT := 400000;
	LCRPID_TUNE_REQU_PER_5 : UDINT := 500000;
	LCRPID_TUNE_REQU_PI : UDINT := 200;
	LCRPID_TUNE_REQU_PID : UDINT := 100;
	LCRPID_TUNE_REQU_STEPRESPONSE : UDINT := 2;
	LCRPID_TUNE_REQU_ZN_DIST : UDINT := 3000;
	LCRPID_TUNE_STATE_CALC_PARA : UINT := 45;
	LCRPID_TUNE_STATE_FINISHED : UINT := 50;
	LCRPID_TUNE_STATE_OSC_CNTLPAR : UINT := 19;
	LCRPID_TUNE_STATE_OSC_PERFORM_1 : UINT := 12;
	LCRPID_TUNE_STATE_OSC_PERFORM_2 : UINT := 13;
	LCRPID_TUNE_STATE_OSC_SEQ_CNTL : UINT := 11;
	LCRPID_TUNE_STATE_OSCILLATE : UINT := 10;
	LCRPID_TUNE_STATE_READY : UINT := 0;
	LCRPID_TUNE_STATE_RESET_CNTL : UINT := 49;
	LCRPID_TUNE_STATE_STEP_MAXGRAD : UINT := 21;
	LCRPID_TUNE_STATE_STEP_WAITEQ1 : UINT := 20;
	LCRPID_TUNE_STATE_STEP_WAITEQ2 : UINT := 22;
	LCRSLIMPID_REQU_CHR_DIST_AP : UDINT := 1000;
	LCRSLIMPID_REQU_CHR_DIST_OS : UDINT := 2000;
	LCRSLIMPID_REQU_CHR_REF_AP : UDINT := 4000;
	LCRSLIMPID_REQU_CHR_REF_OS : UDINT := 5000;
	LCRSLIMPID_REQU_DIR_NEG : UDINT := 20;
	LCRSLIMPID_REQU_DIR_POS : UDINT := 10;
	LCRSLIMPID_REQU_OFF : UDINT := 0;
	LCRSLIMPID_REQU_OSC_1 : UDINT := 10000;
	LCRSLIMPID_REQU_OSC_2 : UDINT := 20000;
	LCRSLIMPID_REQU_OSC_3 : UDINT := 30000;
	LCRSLIMPID_REQU_OSCILLATE : UDINT := 1;
	LCRSLIMPID_REQU_P : UDINT := 300;
	LCRSLIMPID_REQU_PER_3 : UDINT := 300000;
	LCRSLIMPID_REQU_PER_4 : UDINT := 400000;
	LCRSLIMPID_REQU_PER_5 : UDINT := 500000;
	LCRSLIMPID_REQU_PI : UDINT := 200;
	LCRSLIMPID_REQU_PID : UDINT := 100;
	LCRSLIMPID_REQU_READ_PARAS : UDINT := 3;
	LCRSLIMPID_REQU_STEPRESPONSE : UDINT := 2;
	LCRSLIMPID_REQU_WRITE_PARAS : UDINT := 4;
	LCRSLIMPID_REQU_ZN_DIST : UDINT := 3000;
	LCRTEMP_COOL : USINT := 1;
	LCRTEMP_HEAT : USINT := 0;
	LCRTEMP_PT1 : USINT := 0;
	LCRTEMP_PT2 : USINT := 1;
	LCRTEMP_STEP_COOL : UINT := 120;
	LCRTEMP_STEP_DONE : UINT := 130;
	LCRTEMP_STEP_ERROR : UINT := 65535;
	LCRTEMP_STEP_FREE : UINT := 70;
	LCRTEMP_STEP_HEAT : UINT := 30;
	LCRTEMP_STEP_PID : UINT := 80;
	LCRTEMP_STEP_PID_COOL : UINT := 90;
	LCRTEMP_STEP_PID_DONE : UINT := 125;
	LCRTEMP_STEP_PID_DONE_COOLONLY : UINT := 122;
	LCRTEMP_STEP_PID_FREE : UINT := 40;
	LCRTEMP_STEP_START_COOL : UINT := 110;
	LCRTEMP_STEP_START_FREE : UINT := 60;
	LCRTEMP_STEP_START_HEAT : UINT := 20;
	LCRTEMP_STEP_WAIT : UINT := 5;
	LCRTEMP_STEP_WAIT_COOL : UINT := 100;
	LCRTEMP_STEP_WAIT_COOLONLY : UINT := 105;
	LCRTEMP_STEP_WAIT_FREE : UINT := 50;
	LCRTEMP_STEP_WAIT_HEAT : UINT := 10;
	LCRTEMPPID_MODE_AUTO : UDINT := 1;
	LCRTEMPPID_MODE_MAN : UDINT := 2;
	LCRTEMPTune_MODE_DEF : UDINT := 0;
	LCRTEMPTune_MODE_EXP : UDINT := 1;
END_VAR
